// TwinCAT 3 PLC project Sample01
// ProgramVersion: 3.1.4020.10
// libraries:
//   Tc2_Standard, * (Beckhoff Automation GmbH)
//   Tc2_System, * (Beckhoff Automation GmbH)
//   Tc3_Module, * (Beckhoff Automation GmbH)
// project tree:
//   / PlcTask.TcTTO (not stored)
//   POUs/ Class Diagram.TcCD (not stored), FB_AnalogValue.TcPOU, FB_Controller.TcPOU, FB_Lamp.TcPOU (not stored), FB_LampSetDirectDALI.TcPOU, FB_LampOnOffAdapter.TcPOU, FB_LampSetDirectAdapter.TcPOU, FB_LampSetDirectDALIAdapter.TcPOU, FB_LampUpDown.TcPOU, FB_LampSetDirect.TcPOU, FB_LampOnOff.TcPOU, FB_LampUpDownAdapter.TcPOU (not stored), I_Lamp.TcIO (not stored), I_Observer.TcIO, I_Subject.TcIO (not stored), MAIN.TcPOU
// real-time tasks:
//   TASK PlcTask: cycle T#10ms, priority 20, ADS port 350

// ---- POUs/I_Observer.TcIO
INTERFACE I_Observer EXTENDS __System.IQueryInterface

METHOD Update
VAR_INPUT
	nNewValue		: BYTE;
END_VAR
END_METHOD

END_INTERFACE

// ---- POUs/FB_AnalogValue.TcPOU
FUNCTION_BLOCK PUBLIC FB_AnalogValue IMPLEMENTS I_Observer
VAR_INPUT
END_VAR
VAR_OUTPUT
END_VAR
VAR
	_nActualValue		: BYTE;
END_VAR

{attribute 'monitoring' := 'call'}
PROPERTY PUBLIC nValue : BYTE
GET
nValue := _nActualValue;
END_GET
END_PROPERTY

METHOD Update
VAR_INPUT
	nNewValue		: BYTE;
END_VAR
_nActualValue := nNewValue;
END_METHOD

END_FUNCTION_BLOCK

// ---- POUs/FB_Controller.TcPOU
FUNCTION_BLOCK PUBLIC FB_Controller
VAR
	fbActualValue		: FB_AnalogValue;
	_refActiveLamp		: REFERENCE TO FB_Lamp;
END_VAR

// Reduces the control value by 5 in the range of 10 to 100.
METHOD PUBLIC DimDown
IF (__ISVALIDREF(_refActiveLamp)) THEN
	_refActiveLamp.DimDown();
END_IF
END_METHOD

// Increments the control value by 5 in the range of 10 to 100.
METHOD PUBLIC DimUp
IF (__ISVALIDREF(_refActiveLamp)) THEN
	_refActiveLamp.DimUp();
END_IF
END_METHOD

// Sets the control value to 0.
METHOD PUBLIC Off
IF (__ISVALIDREF(_refActiveLamp)) THEN
	_refActiveLamp.Off();
END_IF
END_METHOD

// Sets the control value to 100.
METHOD PUBLIC On
IF (__ISVALIDREF(_refActiveLamp)) THEN
	_refActiveLamp.On();
END_IF
END_METHOD

{attribute 'monitoring' := 'call'}
PROPERTY PUBLIC refActiveLamp : REFERENCE TO FB_Lamp
GET
refActiveLamp REF= _refActiveLamp;
END_GET
SET
IF (__ISVALIDREF(_refActiveLamp)) THEN
	_refActiveLamp.Detach();
END_IF

_refActiveLamp REF= refActiveLamp;

IF (__ISVALIDREF(refActiveLamp)) THEN
	refActiveLamp.Attach(fbActualValue);
END_IF
END_SET
END_PROPERTY

END_FUNCTION_BLOCK

// ---- POUs/FB_LampSetDirectDALI.TcPOU
FUNCTION_BLOCK PUBLIC FB_LampSetDirectDALI EXTENDS FB_LampSetDirect
VAR
END_VAR

// Sets the control value of the DALI lamp to a value between 0 and 254.
METHOD PUBLIC SetLightLevel
VAR_INPUT
	nNewLightLevel		: BYTE(0..254);
END_VAR
nLightLevel := nNewLightLevel;
END_METHOD

END_FUNCTION_BLOCK

// ---- POUs/FB_LampSetDirect.TcPOU
FUNCTION_BLOCK PUBLIC FB_LampSetDirect
VAR
	nLightLevel			: BYTE;
END_VAR

// Sets the control value to a value between 0 and 100.
METHOD PUBLIC SetLightLevel
VAR_INPUT
	nNewLightLevel		: BYTE(0..100);
END_VAR
nLightLevel := nNewLightLevel;
END_METHOD

END_FUNCTION_BLOCK

// ---- POUs/FB_LampOnOffAdapter.TcPOU
FUNCTION_BLOCK PUBLIC FB_LampOnOffAdapter EXTENDS FB_Lamp 
VAR
	fbLampOnOff			: FB_LampOnOff;
END_VAR

// Reduces the control value by 5 in the range of 10 to 100.
METHOD PUBLIC DimDown
fbLampOnOff.DimDown();
IF (_ipObserver <> 0) THEN
	_ipObserver.Update(fbLampOnOff.nLightLevel);
END_IF
END_METHOD

// Increments the control value by 5 in the range of 10 to 100.
METHOD PUBLIC DimUp
fbLampOnOff.DimUp();
IF (_ipObserver <> 0) THEN
	_ipObserver.Update(fbLampOnOff.nLightLevel);
END_IF
END_METHOD

// Sets the control value to 0.
METHOD PUBLIC Off
fbLampOnOff.Off();
IF (_ipObserver <> 0) THEN
	_ipObserver.Update(fbLampOnOff.nLightLevel);
END_IF
END_METHOD

// Sets the control value to 100.
METHOD PUBLIC On
fbLampOnOff.On();
IF (_ipObserver <> 0) THEN
	_ipObserver.Update(fbLampOnOff.nLightLevel);
END_IF
END_METHOD

END_FUNCTION_BLOCK

// ---- POUs/FB_LampOnOff.TcPOU
FUNCTION_BLOCK PUBLIC FB_LampOnOff 
VAR
	nLightLevel			: BYTE;
END_VAR

// Reduces the control value by 5 in the range of 10 to 100.
METHOD PUBLIC DimDown
Off();
END_METHOD

// Increments the control value by 5 in the range of 10 to 100.
METHOD PUBLIC DimUp
On();
END_METHOD

// Sets the control value to 0.
METHOD PUBLIC Off
nLightLevel := 0;
END_METHOD

// Sets the control value to 100.
METHOD PUBLIC On
nLightLevel := 100;
END_METHOD

END_FUNCTION_BLOCK

// ---- POUs/FB_LampSetDirectAdapter.TcPOU
FUNCTION_BLOCK PUBLIC FB_LampSetDirectAdapter EXTENDS FB_Lamp
VAR
	fbLampSetDirect		: FB_LampSetDirect;
END_VAR

// Reduces the control value by 5 in the range of 10 to 100.
METHOD PUBLIC DimDown
IF (fbLampSetDirect.nLightLevel >= 15) THEN
	fbLampSetDirect.SetLightLevel(fbLampSetDirect.nLightLevel - 5);
END_IF
IF (_ipObserver <> 0) THEN
	_ipObserver.Update(fbLampSetDirect.nLightLevel);
END_IF
END_METHOD

// Increments the control value by 5 in the range of 10 to 100.
METHOD PUBLIC DimUp
IF (fbLampSetDirect.nLightLevel <= 95) THEN
	fbLampSetDirect.SetLightLevel(fbLampSetDirect.nLightLevel + 5);
END_IF
IF (_ipObserver <> 0) THEN
	_ipObserver.Update(fbLampSetDirect.nLightLevel);
END_IF
END_METHOD

// Sets the control value to 0.
METHOD PUBLIC Off
fbLampSetDirect.SetLightLevel(0);
IF (_ipObserver <> 0) THEN
	_ipObserver.Update(fbLampSetDirect.nLightLevel);
END_IF
END_METHOD

// Sets the control value to 100.
METHOD PUBLIC On
fbLampSetDirect.SetLightLevel(100);
IF (_ipObserver <> 0) THEN
	_ipObserver.Update(fbLampSetDirect.nLightLevel);
END_IF
END_METHOD

END_FUNCTION_BLOCK

// ---- POUs/FB_LampSetDirectDALIAdapter.TcPOU
FUNCTION_BLOCK PUBLIC FB_LampSetDirectDALIAdapter EXTENDS FB_Lamp
VAR
	fbLampSetDirectDALI		: FB_LampSetDirectDALI;
END_VAR

// Reduces the control value by 5 in the range of 10 to 254.
METHOD PUBLIC DimDown
IF (fbLampSetDirectDALI.nLightLevel >= 15) THEN
	fbLampSetDirectDALI.SetLightLevel(fbLampSetDirectDALI.nLightLevel - 5);
END_IF
IF (_ipObserver <> 0) THEN
	_ipObserver.Update(fbLampSetDirectDALI.nLightLevel);
END_IF
END_METHOD

// Increments the control value by 5 in the range of 10 to 254.
METHOD PUBLIC DimUp
IF (fbLampSetDirectDALI.nLightLevel <= 249) THEN
	fbLampSetDirectDALI.SetLightLevel(fbLampSetDirectDALI.nLightLevel + 5);
END_IF
IF (_ipObserver <> 0) THEN
	_ipObserver.Update(fbLampSetDirectDALI.nLightLevel);
END_IF
END_METHOD

// Sets the control value to 0.
METHOD PUBLIC Off
fbLampSetDirectDALI.SetLightLevel(0);
IF (_ipObserver <> 0) THEN
	_ipObserver.Update(fbLampSetDirectDALI.nLightLevel);
END_IF
END_METHOD

// Sets the control value to 254.
METHOD PUBLIC On
fbLampSetDirectDALI.SetLightLevel(254);
IF (_ipObserver <> 0) THEN
	_ipObserver.Update(fbLampSetDirectDALI.nLightLevel);
END_IF
END_METHOD

END_FUNCTION_BLOCK

// ---- POUs/FB_LampUpDown.TcPOU
FUNCTION_BLOCK FB_LampUpDown
VAR
	nLightLevel			: BYTE;	
END_VAR

// Reduces the control value by 1 in the range of 10 to 100. 
METHOD PUBLIC OneStepDown
nLightLevel := nLightLevel - 1;
IF (nLightLevel < 10) THEN
	nLightLevel := 10;
END_IF
END_METHOD

// Increments the control value by 1 in the range of 10 to 100.
METHOD PUBLIC OneStepUp
nLightLevel := nLightLevel + 1;
IF (nLightLevel > 100) THEN
	nLightLevel := 100;
END_IF
END_METHOD

// Toggles the control value between 0 and 100.
METHOD PUBLIC OnOff
IF (nLightLevel > 0) THEN
	nLightLevel := 0;
ELSE
	nLightLevel := 100;
END_IF
END_METHOD

END_FUNCTION_BLOCK

// ---- POUs/MAIN.TcPOU
PROGRAM MAIN
VAR
	fbController				: FB_Controller();
	fbLampOnOffAdapter			: FB_LampOnOffAdapter();
	fbLampSetDirectAdapter		: FB_LampSetDirectAdapter();
	fbLampUpDownAdapter			: FB_LampUpDownAdapter();
	fbLampSetDirectDALIAdapter	: FB_LampSetDirectDALIAdapter();	
	nSetLamp					: INT;
	bDimUp, bDimDown			: BOOL;
	bOff, bOn					: BOOL;
	nLightLevel					: BYTE;
END_VAR

CASE nSetLamp OF
	1:
		fbController.refActiveLamp REF= fbLampOnOffAdapter;
		nSetLamp := 0;
	2:
		fbController.refActiveLamp REF= fbLampSetDirectAdapter;
		nSetLamp := 0;
	3:
		fbController.refActiveLamp REF= fbLampUpDownAdapter;
		nSetLamp := 0;
	4:
		fbController.refActiveLamp REF= fbLampSetDirectDALIAdapter;
		nSetLamp := 0;
END_CASE

nLightLevel := fbController.fbActualValue.nValue;

IF (bDimUp) THEN
	fbController.DimUp();
	bDimUp := FALSE;
END_IF

IF (bDimDown) THEN
	fbController.DimDown();
	bDimDown := FALSE;
END_IF

IF (bOff) THEN
	fbController.Off();
	bOff := FALSE;
END_IF

IF (bOn) THEN
	fbController.On();
	bOn := FALSE;
END_IF

END_PROGRAM
